PROGRAM Axis04_Command
VAR
//SysTem_Bit
	Always_ON	:	BOOL	:=TRUE	;//상시 ON
	Always_OFF	:	BOOL	:=FALSE	;//상시 OFF
//Motor_Command
	Axis04: AXIS_REF;											//회전축
	Axis04_MC_Power: MC_Power;
	Axis04_MC_Home: FB_HomeBeforeMoveAX8000:=(channel:=2);
	Axis04_Jog: MC_Jog;
	Axis04_Home_Pos_Move: MC_MoveAbsolute;
	Axis04_Wait_Pos_Move: MC_MoveAbsolute;
	Axis04_Target_Pos_Move: MC_MoveAbsolute;
	Axis04_Work_End_Move: MC_MoveAbsolute;
	Axis04_Maint_Move: MC_MoveAbsolute;
	Axis04_Tool_Change_Move: MC_MoveAbsolute;
	Axis04_Mastering_Move: MC_MoveAbsolute;	
	
	Axis04_Calibration_Move: MC_MoveAbsolute;
	
	Axis04_Work_Torque: MC_TorqueControl;
	Axis04_Work_Torque2: MC_TorqueControl;
	Options: ST_TorqueControlOptions;
	Timer03: TON;
	Axis04_Cleaning_Pos_Move: MC_MoveAbsolute;
	keb_Z: BOOL;
	Keb_Z_data_PB: BOOL;
END_VAR

VAR_INPUT
	MC_Return_Move: MC_MoveAbsolute;
END_VAR
VAR // added by the converter: edge detectors and wires of the graphical bodies
    _rt1, _rt2 : R_TRIG;
END_VAR

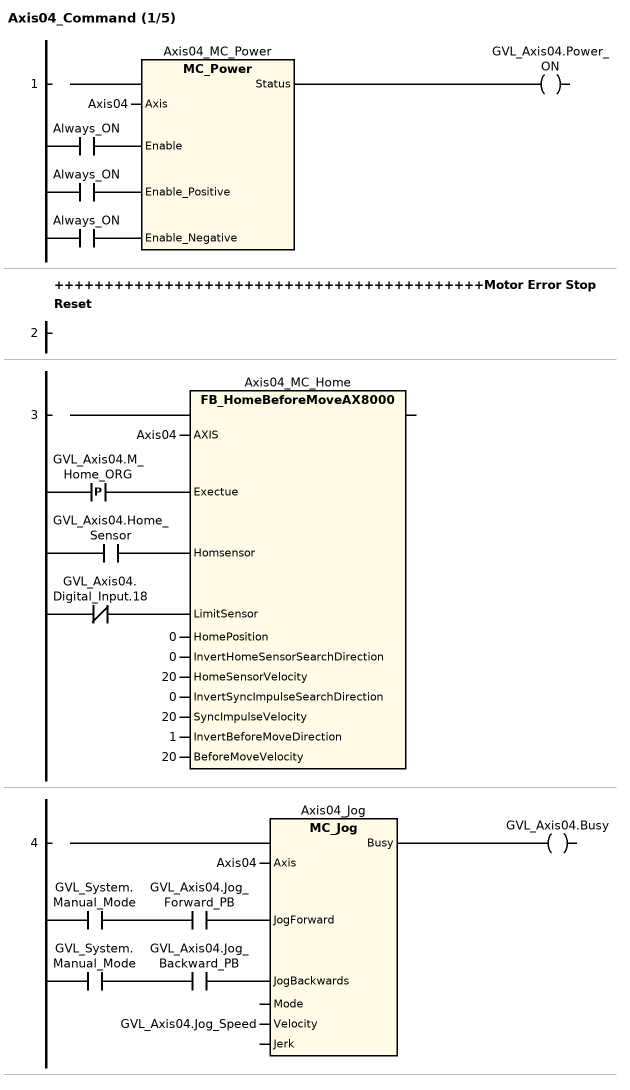
// NETWORK 1
Axis04_MC_Power(
    Axis := Axis04,
    Enable := Always_ON,
    Enable_Positive := Always_ON,
    Enable_Negative := Always_ON); // MC_Power
GVL_Axis04.Power_ON := Axis04_MC_Power.Status;

// NETWORK 2: +++++++++++++++++++++++++++++++++++++++++++Motor Error Stop Reset

// NETWORK 3
_rt1(CLK := GVL_Axis04.M_Home_ORG);
Axis04_MC_Home(
    AXIS := Axis04,
    Exectue := _rt1.Q,
    Homsensor := GVL_Axis04.Home_Sensor,
    LimitSensor := NOT GVL_Axis04.Digital_Input.18,
    HomePosition := 0,
    InvertHomeSensorSearchDirection := 0,
    HomeSensorVelocity := 20,
    InvertSyncImpulseSearchDirection := 0,
    SyncImpulseVelocity := 20,
    InvertBeforeMoveDirection := 1,
    BeforeMoveVelocity := 20); // FB_HomeBeforeMoveAX8000

// NETWORK 4
Axis04_Jog(
    Axis := Axis04,
    JogForward := GVL_System.Manual_Mode AND GVL_Axis04.Jog_Forward_PB,
    JogBackwards := GVL_System.Manual_Mode AND GVL_Axis04.Jog_Backward_PB,
    Velocity := GVL_Axis04.Jog_Speed,
    Busy => GVL_Axis04.Busy); // MC_Jog

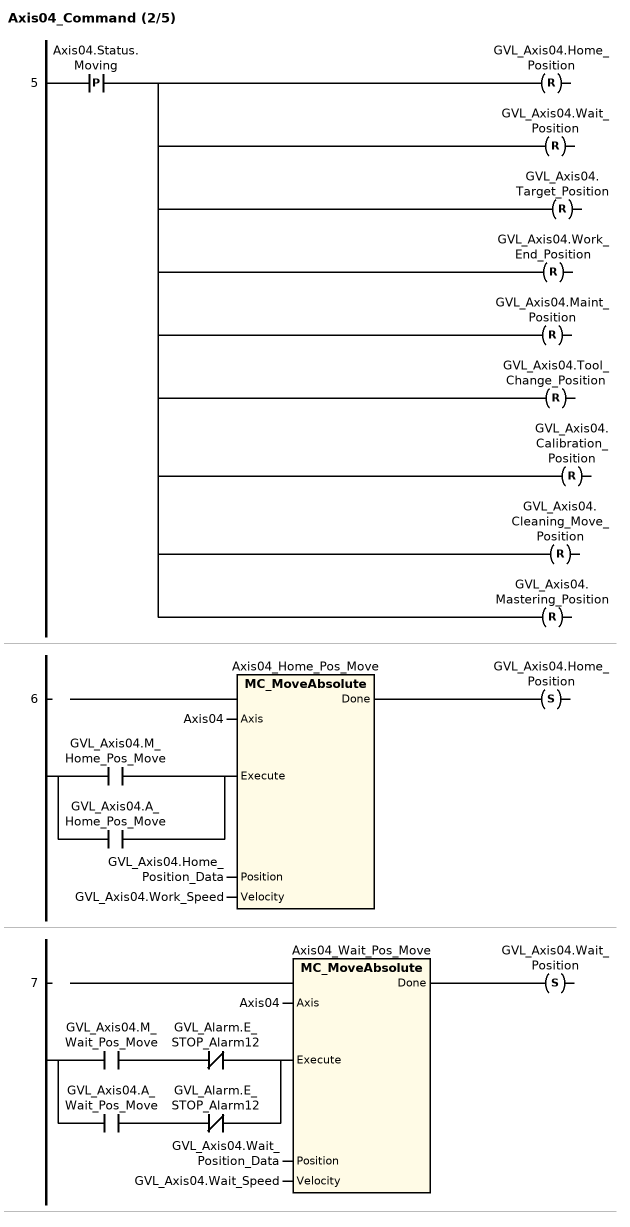
// NETWORK 5
_rt2(CLK := Axis04.Status.Moving);
GVL_Axis04.Home_Position R= _rt2.Q;
GVL_Axis04.Wait_Position R= _rt2.Q;
GVL_Axis04.Target_Position R= _rt2.Q;
GVL_Axis04.Work_End_Position R= _rt2.Q;
GVL_Axis04.Maint_Position R= _rt2.Q;
GVL_Axis04.Tool_Change_Position R= _rt2.Q;
GVL_Axis04.Calibration_Position R= _rt2.Q;
GVL_Axis04.Cleaning_Move_Position R= _rt2.Q;
GVL_Axis04.Mastering_Position R= _rt2.Q;

// NETWORK 6
Axis04_Home_Pos_Move(
    Axis := Axis04,
    Execute := GVL_Axis04.M_Home_Pos_Move OR GVL_Axis04.A_Home_Pos_Move,
    Position := GVL_Axis04.Home_Position_Data,
    Velocity := GVL_Axis04.Work_Speed); // MC_MoveAbsolute
GVL_Axis04.Home_Position S= Axis04_Home_Pos_Move.Done;

// NETWORK 7
Axis04_Wait_Pos_Move(
    Axis := Axis04,
    Execute := GVL_Axis04.M_Wait_Pos_Move AND NOT GVL_Alarm.E_STOP_Alarm12 OR GVL_Axis04.A_Wait_Pos_Move AND NOT GVL_Alarm.E_STOP_Alarm12,
    Position := GVL_Axis04.Wait_Position_Data,
    Velocity := GVL_Axis04.Wait_Speed); // MC_MoveAbsolute
GVL_Axis04.Wait_Position S= Axis04_Wait_Pos_Move.Done;

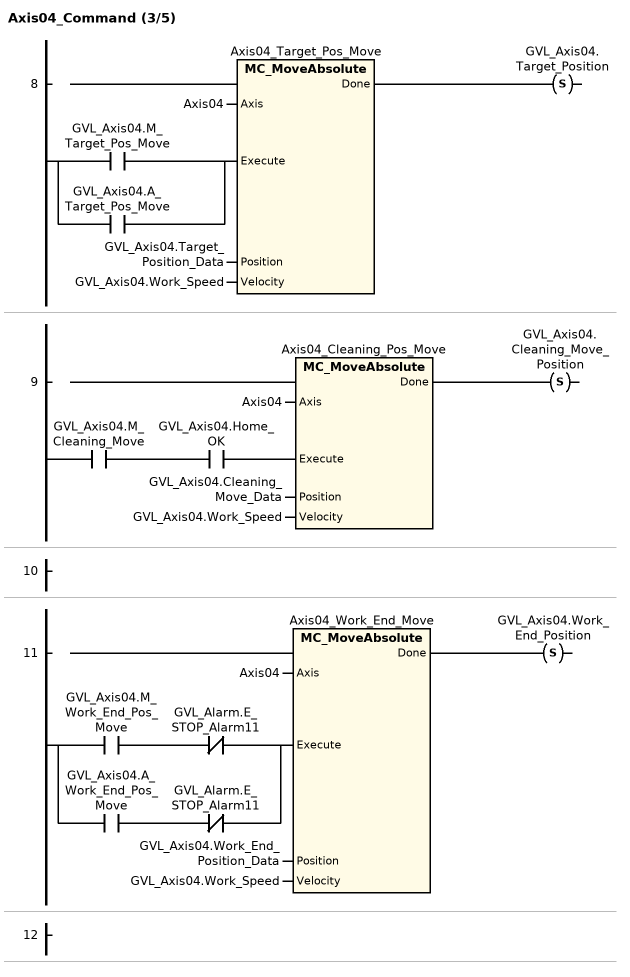
// NETWORK 8
Axis04_Target_Pos_Move(
    Axis := Axis04,
    Execute := GVL_Axis04.M_Target_Pos_Move OR GVL_Axis04.A_Target_Pos_Move,
    Position := GVL_Axis04.Target_Position_Data,
    Velocity := GVL_Axis04.Work_Speed); // MC_MoveAbsolute
GVL_Axis04.Target_Position S= Axis04_Target_Pos_Move.Done;

// NETWORK 9
Axis04_Cleaning_Pos_Move(
    Axis := Axis04,
    Execute := GVL_Axis04.M_Cleaning_Move AND GVL_Axis04.Home_OK,
    Position := GVL_Axis04.Cleaning_Move_Data,
    Velocity := GVL_Axis04.Work_Speed); // MC_MoveAbsolute
GVL_Axis04.Cleaning_Move_Position S= Axis04_Cleaning_Pos_Move.Done;

// NETWORK 10

// NETWORK 11
Axis04_Work_End_Move(
    Axis := Axis04,
    Execute := GVL_Axis04.M_Work_End_Pos_Move AND NOT GVL_Alarm.E_STOP_Alarm11 OR GVL_Axis04.A_Work_End_Pos_Move AND NOT GVL_Alarm.E_STOP_Alarm11,
    Position := GVL_Axis04.Work_End_Position_Data,
    Velocity := GVL_Axis04.Work_Speed); // MC_MoveAbsolute
GVL_Axis04.Work_End_Position S= Axis04_Work_End_Move.Done;

// NETWORK 12

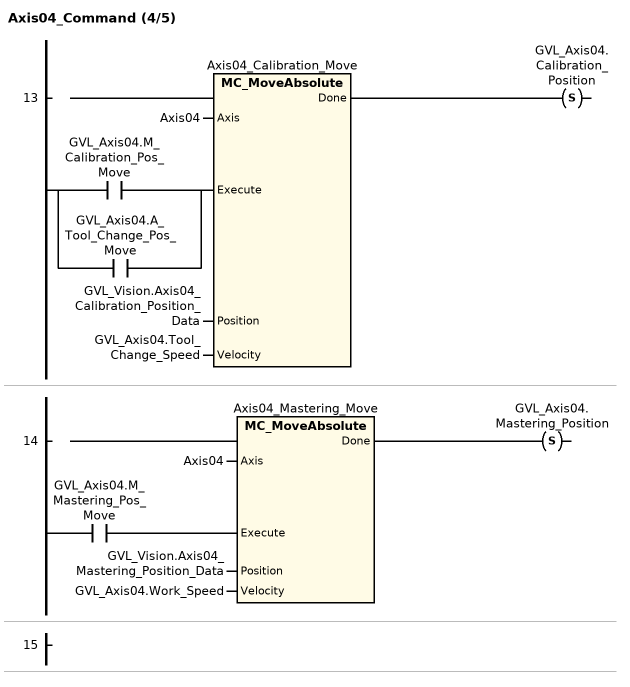
// NETWORK 13
Axis04_Calibration_Move(
    Axis := Axis04,
    Execute := GVL_Axis04.M_Calibration_Pos_Move OR GVL_Axis04.A_Tool_Change_Pos_Move,
    Position := GVL_Vision.Axis04_Calibration_Position_Data,
    Velocity := GVL_Axis04.Tool_Change_Speed); // MC_MoveAbsolute
GVL_Axis04.Calibration_Position S= Axis04_Calibration_Move.Done;

// NETWORK 14
Axis04_Mastering_Move(
    Axis := Axis04,
    Execute := GVL_Axis04.M_Mastering_Pos_Move,
    Position := GVL_Vision.Axis04_Mastering_Position_Data,
    Velocity := GVL_Axis04.Work_Speed); // MC_MoveAbsolute
GVL_Axis04.Mastering_Position S= Axis04_Mastering_Move.Done;

// NETWORK 15

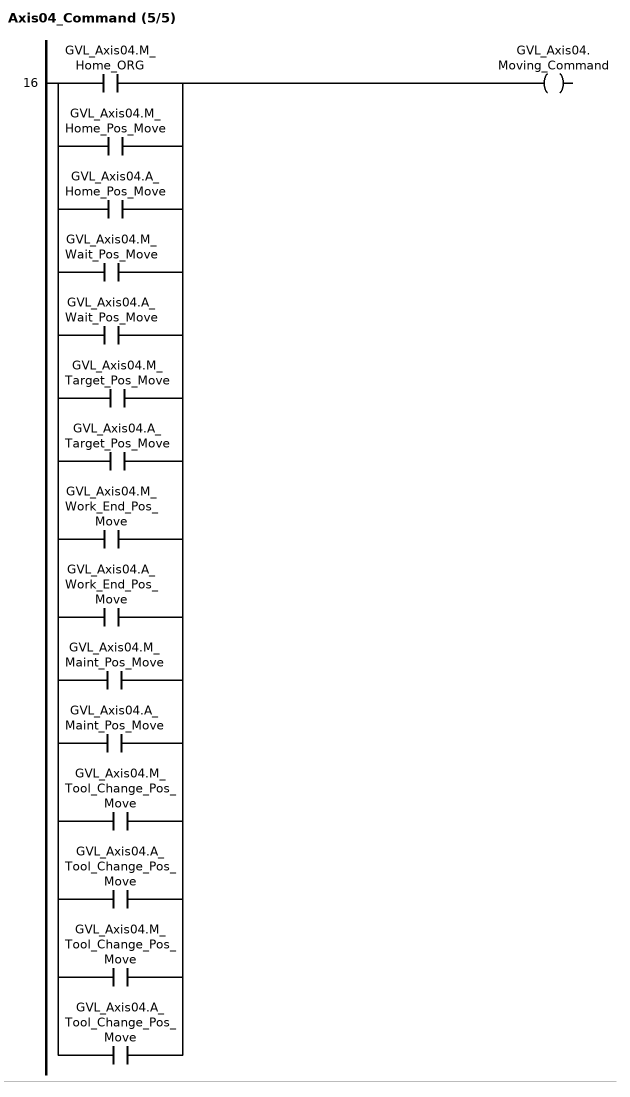
// NETWORK 16
GVL_Axis04.Moving_Command := GVL_Axis04.M_Home_ORG OR GVL_Axis04.M_Home_Pos_Move OR GVL_Axis04.A_Home_Pos_Move OR GVL_Axis04.M_Wait_Pos_Move OR GVL_Axis04.A_Wait_Pos_Move OR GVL_Axis04.M_Target_Pos_Move OR GVL_Axis04.A_Target_Pos_Move OR GVL_Axis04.M_Work_End_Pos_Move OR GVL_Axis04.A_Work_End_Pos_Move OR GVL_Axis04.M_Maint_Pos_Move OR GVL_Axis04.A_Maint_Pos_Move OR GVL_Axis04.M_Tool_Change_Pos_Move OR GVL_Axis04.A_Tool_Change_Pos_Move OR GVL_Axis04.M_Tool_Change_Pos_Move OR GVL_Axis04.A_Tool_Change_Pos_Move;

END_PROGRAM

(* stored: Version 1.1.0.1, ProductVersion 3.1.4024.16
   POU Axis04_Command: Id {cc8fb3d6-0882-4df8-adca-47558e6aac56}, SpecialFunc None *)
